FUNCTION_BLOCK FB_DriveCAN EXTENDS FB_DriveBase
VAR_INPUT
END_VAR
VAR_OUTPUT
END_VAR
VAR
END_VAR

METHOD Disable : BOOL
END_METHOD

METHOD Enable : BOOL
END_METHOD

METHOD MoveToPosition : BOOL
END_METHOD

METHOD Reset : BOOL
END_METHOD

END_FUNCTION_BLOCK

(* stored: Version 1.1.0.1, ProductVersion 3.1.4024.6
   POU FB_DriveCAN: Id {f9c6364f-4df9-4b94-af6b-0e9da0626e79}, SpecialFunc None
   Method Disable: Id {0725cec4-162a-4e4c-8bb9-5063bf747a27}
   Method Enable: Id {651f9e9b-28ad-4e59-91bd-bdb4d3b24d2f}
   Method MoveToPosition: Id {c21be33c-c4f2-4da8-835d-7117a3f37cee}
   Method Reset: Id {f6b2a70a-37d6-47c6-a94f-28b2773cb345} *)
